FUNCTION_BLOCK ActuatorMonitor
VAR_INPUT
	Output: LREAL;
	Input: LREAL;
	Activated: BOOL := TRUE;
	ActivatedError: BOOL := FALSE;
	TimeoutMs: DINT := 30000;
	Treshold: LREAL := 0.1;
END_VAR
VAR_OUTPUT
	Error: BOOL := FALSE;
END_VAR
VAR
	ActivatedSignal: DigitalSignal;
	OutputOnTimer: Timer;
	InputOffTimer: Timer;
END_VAR

// Measure ON time for activation signal
ActivatedSignal(Signal := Activated);

// Measure ON time for output signal
IF Output < Treshold THEN
	OutputOnTimer.Restart();
END_IF

// Measure OFF time for 50% input signal
IF Input >= (Treshold / 2) THEN
	InputOffTimer.Restart();
END_IF

Error := 	(
				(ActivatedSignal.OnTime() > TimeoutMs) AND 
				(OutputOnTimer.ElapsedTime() > TimeoutMs) AND 
				(
					(InputOffTimer.ElapsedTime() > TimeoutMs) OR
					ActivatedError
				)
			);

END_FUNCTION_BLOCK

(* stored: Version 1.1.0.1, ProductVersion 3.1.4024.3
   POU ActuatorMonitor: Id {0cd89761-dd24-4a1e-8b25-84bc93830cf6}, SpecialFunc None *)
